(*
SPDX-FileCopyrightText: © 2026 Oleksandr Tiutyk <trofimich@gmail.com>
SPDX-License-Identifier: MIT
License: https://opensource.org/license/mit
*)

(*!
<summary>Exposes the compiler-initialized namespace of Collections.</summary>
<description>
Internal metadata provider; Name borrows the extractor string and must not be modified. Do not execute this
program explicitly.
</description>
*)

{attribute 'no_explicit_call' := 'do not call this POU directly'}
PROGRAM INTERNAL CurrentNamespace
VAR
	{attribute 'hide'} 
	_NamespaceExtractor : NamespaceExtractor;
END_VAR

(*!
<summary>Borrows the compiler-initialized namespace string.</summary>
<description>
Read-only metadata backed by NamespaceExtractor; callers must not modify it.
</description>
*)
{attribute 'monitoring' := 'call'}
PROPERTY Name : REFERENCE TO STRING
GET
Name REF= _NamespaceExtractor.CurrentNamespace;
END_GET
END_PROPERTY

END_PROGRAM

(* stored: Version 1.1.0.1
   POU CurrentNamespace: Id {d0d30f2d-b5ef-411b-a26a-5471b49c1d92}, SpecialFunc None
   Property Name: Id {d81efea1-8190-4909-bfda-0451a9113803}
   Get Get: Id {0aa210e0-fb32-4a5b-bdad-8914a0728202} *)
